// TIA Portal V19 export
DATA_BLOCK "GlobalData"   // DB6
{ S7_Optimized_Access := 'TRUE' }
// stored: MemoryReserve 100
   VAR
      UnixTimestamp : DInt;
      SensorsSimulation : "typeSimSensors";
      StatesSimulation { S7_SetPoint := 'True'} : "typeSimStates";
   END_VAR
BEGIN
END_DATA_BLOCK
